FUNCTION_BLOCK SimpleClamp
VAR_INPUT
	ClampRequest : BOOL;
	UnClampRequest : BOOL;
	Limit_NC_NO_CI : BOOL;	// Using NC limit switches =0; Using NO Limit switches =1;
	
END_VAR
VAR_OUTPUT
	
	Clamped : BOOL;
	Unclamped : BOOL;
END_VAR
VAR
	
	//HLFB_FI 			AT %I*	: BOOL;	//high level feedback 
	
	Enable_FO 				AT %Q*  : BOOL;		//Enable ClearPath
	InputAOutCW_FO  		AT %Q* 	: BOOL; 	//input A of clearpath motor, Clockwise request move output from plc
	InputBOutCCW_FO  		AT %Q* 	: BOOL; 	//input B of clearpath motor, CounterClockwise move output from plc
	
	ClampedSensorInput_FI 	AT %I* : BOOL; 
	UnclampedSensorInput_FI AT %I* : BOOL; 
	

	
END_VAR



//Move requests if limit switches are NC

IF Limit_NC_NO_CI = 0 THEN
	IF ClampRequest AND ClampedSensorInput_FI THEN
		Enable_FO := 1;
		InputBOutCCW_FO := 1; //Clamp Direction
	ELSE
		ClampRequest := 0;
	END_IF
	
	IF UnclampRequest AND UnclampedSensorInput_FI THEN
		Enable_FO := 1;
		InputAOutCW_FO := 1; //unClamp Direction
	ELSE
		UnclampRequest :=0;
	END_IF
	
	IF NOT(UnclampRequest) AND NOT(ClampRequest) THEN
		Enable_FO := 0;
		InputAOutCW_FO := 0; //unClamp Direction
		InputBOutCCW_FO := 0; //Clamp Direction
	END_IF
	
	//FB OUTPUTS
	IF NOT(ClampedSensorInput_FI) THEN
		Clamped := 1;
	ELSE
		Clamped := 0;
	END_IF
	
	
	IF NOT(UnclampedSensorInput_FI) THEN
		Unclamped := 1;
	ELSE
		Unclamped := 0;
	END_IF
	
END_IF

END_FUNCTION_BLOCK

(* stored: Version 1.1.0.1, ProductVersion 3.1.4024.12
   POU SimpleClamp: Id {1dc743ec-aa17-4723-bc6d-41ebab479e0a}, SpecialFunc None *)
